(* IEC 61131-3 sources: Std_PalletMover/Class/CanOpenCyncMaster, 1 file *)

(* ---- CanOpenCyncMaster.st ---- *)
(*!
<Class
	Name               = "CanOpenCyncMaster"
	Revision           = "0.0"
	RealtimeTask       = "true"
	DefRealtime        = "100 ms"
	CyclicTask         = "false"
	BackgroundTask     = "false"
	Sigmatek           = "false"
	OSInterface        = "false"
	HighPriority       = "false"
	Automatic          = "false"
	UpdateMode         = "Prescan"
	SharedCommandTable = "true"
	Objectsize         = "(480,360)">
	<Channels>
		<Server Name="ClassSvr" Visualized="false" Initialize="false" WriteProtected="false" Retentive="false"/>
		<Server Name="HeartbeatTime" Visualized="true" Initialize="true" DefValue="1000" WriteProtected="false" Retentive="SRam" Comment="[ms]"/>
		<Client Name="CanOpen" Required="true" Internal="true"/>
		<Client Name="cNode" Required="true" Internal="false"/>
		<Client Name="Driver" Required="false" Internal="false"/>
	</Channels>
	<Network Name="CanOpenCyncMaster">
		<!-- List of Components in this network -->
		<Components>
			<Object
				Name       = "CanOpen"
				Class      = "CanOpenBase"
				Position   = "(210,120)"
				Visualized = "true"
				CyclicTime = "10 ms">
				<Channels>
					<Server Name="Server0"/>
					<Client Name="cNode" Value="1"/>
					<Client Name="ConfigData"/>
					<Client Name="Driver"/>
				</Channels>
			</Object>
		</Components>
		<Comments>
		</Comments>
		<!-- List of Connections in this network -->
		<Connections>
			<Connection Source="this.CanOpen" Destination="CanOpen.Server0"/>
			<Connection Source="CanOpen.Driver" Destination="this.Driver" Vertices="(210,210),(38,210),"/>
			<Connection Source="CanOpen.cNode" Destination="this.cNode" Vertices="(210,270),(38,270),"/>
		</Connections>
		<!-- Headerfiles -->
		<Options>
		</Options>
	</Network>
</Class>
*)
CanOpenCyncMaster : CLASS
	TYPE
	  NMT_Commands :  //! <Type Public="true" Name="NMT_Commands"/>
	  (
	    NC_Start:=1,
	    NC_Stop:=2,
	    NC_GotoPreOperational:=128,
	    NC_Reset:=129,
	    NC_ResetComm:=130
	  )$DINT;
	END_TYPE
  //Servers:
	ClassSvr 	: SvrChCmd_DINT;
	HeartbeatTime 	: SvrCh_UDINT;
  //Clients:
	Driver 	: CltChCmd_CanDriverBase;
	cNode 	: CltCh_DINT;
	CanOpen 	: CltChCmd_CanOpenBase;
  //Variables:
		Stepper 	: DINT;
		tHeartbeat 	: UDINT;
  //Functions:

	FUNCTION VIRTUAL GLOBAL RtWork
		VAR_INPUT
			EAX 	: UDINT;
		END_VAR
		VAR_OUTPUT
			state (EAX) 	: UDINT;
		END_VAR;
  //Tables:
	FUNCTION @STD
		VAR_OUTPUT
			ret_code	: CONFSTATES;
		END_VAR;
	FUNCTION GLOBAL TAB @CT_;
END_CLASS;

#pragma using CanOpenBase
#pragma usingLtd CanDriverBase

FUNCTION VIRTUAL GLOBAL CanOpenCyncMaster::RtWork
	VAR_INPUT
		EAX 	: UDINT;
	END_VAR
	VAR_OUTPUT
		state (EAX) 	: UDINT;
	END_VAR

  VAR
  	retval : dint;
  END_VAR

  IF IsClientConnected(#Driver) = 0 THEN
	  state := READY;
    RETURN;
  END_IF;

  retval := CanOpen.BuildSync(SyncId:=128);

  retval := CanOpen.BuildNmt(NmtId:=0, Cmnd:=01, Node:=0);

  CASE Stepper OF
    0:
    CanOpen.BuildHeartbeat();
     tHeartbeat := ops.tAbsolute;

     Stepper += 1;

    1:
     if ops.tAbsolute - tHeartbeat > HeartbeatTime then
       Stepper -= 1;
     end_if;

    END_CASE;

	state := READY;

END_FUNCTION
